PROGRAM MAIN_ST01
VAR
	fbStation01							: RACBaseObjects.FB_Station;
	fbConveyor							: RACBaseObjects.FB_Conveyor;
	fbControllerSupply					: FB_ControllerSupply;
	fbBatterySupply						: FB_BatterySupply;
	fbEndcapAsm							: FB_EndcapAsm;
	fbControllerAsm						: FB_ControllerAsm;
	fbLoadStation						: FB_LoadStation;
END_VAR

	fbStation01(bInitFinished:=fbControllerSupply.bInit_Finished AND fbBatterySupply.bInit_Finished AND fbConveyor.bInit_Finished);

	fbConveyor(							sDeviceID:='',
										bStopExecution:=fbStation01.bStop,
										bAlarmReset:=fbStation01.bAlarmReset,
										diStationState:=fbStation01.diStationState,
										bInit_StartPermissive:=TRUE,
										bIn_SafeToMove:=FALSE,
										bIn_AllProcessComplete:=FALSE,
										lrDistance:=0,
										lrOffsetPos:=0,
										bIn_IsClamped:=FALSE,
										bIn_IsUnclamped:=FALSE);
										
	fbLoadStation(						sDeviceID:='',
										bStopExecution:=fbStation01.bStop,
										bAlarmReset:=fbStation01.bAlarmReset,
										diStationState:=fbStation01.diStationState,
										bInit_StartPermissive := TRUE,
										bDisableScan := TRUE,
										bIn_MovePermisive := FALSE,
										bIn_CvyStepDone := FALSE);

	fbEndcapAsm(						sDeviceID:='',
										bStopExecution:=fbStation01.bStop,
										bAlarmReset:=fbStation01.bAlarmReset,
										diStationState:=fbStation01.diStationState,
										bInit_StartPermissive:=TRUE,
										bSafetyBoxPlace_permissive :=TRUE);
	
										
	fbControllerSupply(					sDeviceID:='',
										bStopExecution:=fbStation01.bStop,
										bAlarmReset:=fbStation01.bAlarmReset,
										diStationState:=fbStation01.diStationState,
										bInit_StartPermissive:=TRUE,
										bSafetyBoxPlace_permissive:=FALSE,
										bPlace_MaterialRequest:=FALSE);
										
	fbControllerAsm(					sDeviceID:='',
										bStopExecution:=fbStation01.bStop,
										bAlarmReset:=fbStation01.bAlarmReset,
										diStationState:=fbStation01.diStationState,
										bInit_StartPermissive:=TRUE,
										sSerialReceived:=fbControllerSupply.sPieceSN,	
										bIn_RailReady:=fbConveyor.bOut_MoveDone);
										
	fbBatterySupply(					sDeviceID:='',
										bStopExecution:=fbStation01.bStop,
										bAlarmReset:=fbStation01.bAlarmReset,
										diStationState:=fbStation01.diStationState,
										bInit_StartPermissive:=TRUE,
										bSafetyBoxPlace_permissive := FALSE,
										bPlace_MaterialRequest := TRUE);

END_PROGRAM

(* stored: Version 1.1.0.1, ProductVersion 3.1.4024.12
   POU MAIN_ST01: Id {9d1691a3-5908-4ed4-af9f-582490a1a007}, SpecialFunc None *)
